TYPE ST_AxisParamSpec :
STRUCT
    eParam: E_AxisParameters;
    fValue: LREAL;
END_STRUCT
END_TYPE

(* stored: Version 1.1.0.1
   DUT ST_AxisParamSpec: Id {786e4eb1-46f0-0178-3b79-82a7fdcac1a2} *)
